(*
Some short description.
*)FUNCTION_BLOCK AutoFunctionBlock
VAR_INPUT
    someInput       : BOOL;         // Important description
END_VAR
VAR_OUTPUT
    someOutput      : BOOL;
END_VAR
VAR
END_VAR

(*
Method description!
*)
METHOD PRIVATE AutoMethod : BOOL;
VAR_INPUT
    methodInput     : UDINT;
END_VAR
END_METHOD

(*
Reference to a variable that might be read-only.
*)
PROPERTY AutoProperty : REFERENCE TO LREAL
GET
END_GET
SET
END_SET
END_PROPERTY

END_FUNCTION_BLOCK

(* stored: Version 1.1.0.1, ProductVersion 3.1.4024.11
   POU AutoFunctionBlock: Id {e9c77de4-fb3d-4077-ade3-01c3e8e43ca3}, SpecialFunc None
   Method AutoMethod: Id {1b9475da-fcfe-487e-a0dd-df8806a0c2df}
   Property AutoProperty: Id {cdcba121-a220-4eb8-8f4d-8924b3a02f60}
   Get Get: Id {fe3cd6e4-aa00-4539-98af-b9fb9586655f}
   Set Set: Id {80addca4-0610-47c4-8a76-38191658e0bd} *)
